// TIA Portal V20 export
DATA_BLOCK "DB_Digital_Output"   // DB3
{ S7_Optimized_Access := 'TRUE' }
// stored: AutoNumber false, MemoryReserve 100
   VAR
      Spin_Carousel_Frequency_Inverter_Speed_1 : Bool;
      Spin_Carousel_Frequency_Inverter_Speed_2 : Bool;
      Spin_Carousel_Frequency_Inverter_Speed_3 : Bool;
      Conveyor_Belt_Frequency_Inverter_Speed_1 : Bool;
      Conveyor_Belt_Frequency_Inverter_Speed_2 : Bool;
      Conveyor_Belt_Frequency_Inverter_Speed_3 : Bool;
      Turn_On_Conveyor_Belt_Motor_Spinner_Get_Entrace_Function_Test : Bool;
      Turn_On_Conveyor_Belt_Motor_Rework_Conveyor_Belt_Get_Entrace_Functional_Test : Bool;
      Turn_On_Conveyor_Belt_Motor_Spinner_Get_Exit_Functional_Test : Bool;
      Turn_On_Conveyor_Belt_Motor_Rework_Conveyor_Belt_Get_Exit_Funcional_Test : Bool;
      Open_Air_Pressure : Bool;
      Valve_Advance_Spinner_Entrace_Functional_Test : Bool;
      Valve_Advance_Spinner_Exit_Functional_Test : Bool;
      Signal_Pre_Functional_Test_Production_Line : Bool;
      Digital_Output_14 : Bool;
      Digital_Output_15 : Bool;
      Digital_Output_16 : Bool;
      Digital_Output_17 : Bool;
      Digital_Output_18 : Bool;
      Digital_Output_19 : Bool;
      Digital_Output_20 : Bool;
      Digital_Output_21 : Bool;
      Digital_Output_22 : Bool;
      Digital_Output_23 : Bool;
      Voltage_220V_Selected : Bool;
      Voltage_127V_Selected : Bool;
   END_VAR
BEGIN
END_DATA_BLOCK
